TYPE Vec8b : ARRAY[1..8] OF BOOl; END_TYPE

(* stored: Version 1.1.0.1, ProductVersion 3.1.4024.11
   DUT Vec8b: Id {54449b61-0ec2-4ccd-8cc5-6cf0710a7522} *)
